(* Logix 5000 project; controller Week1 vendor 1 type 14 code 151 rev 37.11; software revision 37.00 *)

TASK MainTask (continuous, watchdog 500 ms) : MainProgram

MODULES
   Local : vendor 1 type 14 code 151 (Compact 0, rev 37.11)
      Discrete_IO : Embedded (Compact 1, rev 3.1, Output RPI 20 ms)
      Analog_IO : Embedded (Compact 2, rev 1.1, Output RPI 80 ms)
      Counters : Embedded (Compact 3, rev 1.1, Output RPI 20 ms)
END_MODULES

PROGRAM MainProgram   (* main routine MainRoutine *)
VAR
   Cycle_Timer : COUNTER := (PRE := 3, ACC := 3, DN := 1);
   Green_Light : ALIAS FOR Local:1:O.Data.2;
   Green_Pct : REAL := 39.863888;
   Green_Timer : TIMER := (PRE := 300000, ACC := 71755);
   Light_Off : BOOL;
   Logic_Sub : DINT;
   Red_Light : ALIAS FOR Local:1:O.Data.0;
   Red_Pct : REAL := 33.332222;
   Red_Timer : TIMER := (PRE := 300000, ACC := 59998);
   Res_Value : DINT;
   Reset_All : BOOL;
   Reset_PB : ALIAS FOR Local:1:I.Data.0;
   Test_Tag : DINT := 12345;
   Total_Time : DINT;
   Traffic_Timer : TIMER := (PRE := 60000);
   Yellow_Light : ALIAS FOR Local:1:O.Data.1;
   Yellow_Pct : REAL := 8.331667;
   Yellow_Timer : TIMER := (PRE := 300000, ACC := 14997);
END_VAR

ROUTINE MainRoutine   (* ladder *)
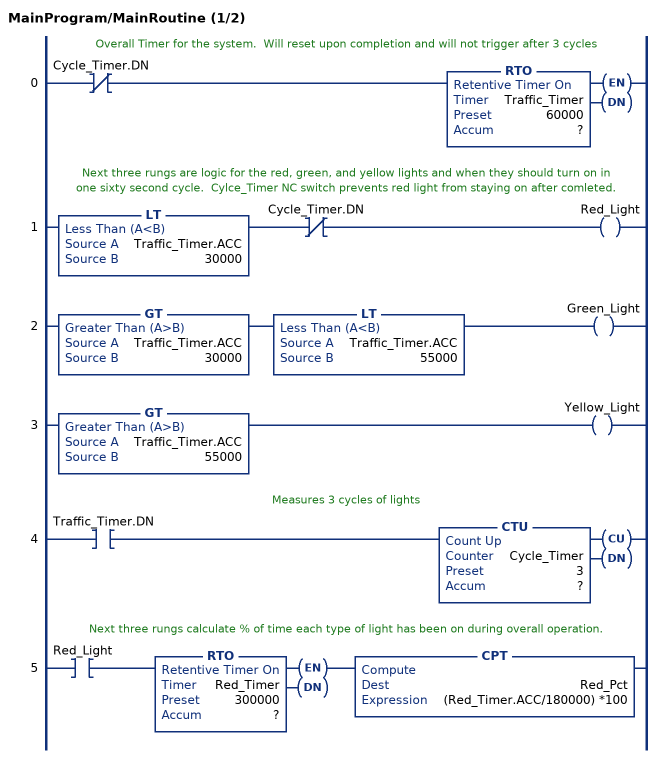
   // Overall Timer for the system.  Will reset upon completion and will not trigger after 3 cycles
   0: XIO(Cycle_Timer.DN)RTO(Traffic_Timer,?,?);
   // Next three rungs are logic for the red, green, and yellow lights and when they should turn on in one sixty second cycle.  Cylce_Timer NC switch prevents red light from staying on after comleted.
   1: LT(Traffic_Timer.ACC,30000)XIO(Cycle_Timer.DN)OTE(Red_Light);
   2: GT(Traffic_Timer.ACC,30000)LT(Traffic_Timer.ACC,55000)OTE(Green_Light);
   3: GT(Traffic_Timer.ACC,55000)OTE(Yellow_Light);
   // Measures 3 cycles of lights
   4: XIC(Traffic_Timer.DN)CTU(Cycle_Timer,?,?);
   // Next three rungs calculate % of time each type of light has been on during overall operation.
   5: XIC(Red_Light)RTO(Red_Timer,?,?)CPT(Red_Pct,(Red_Timer.ACC/180000) *100);
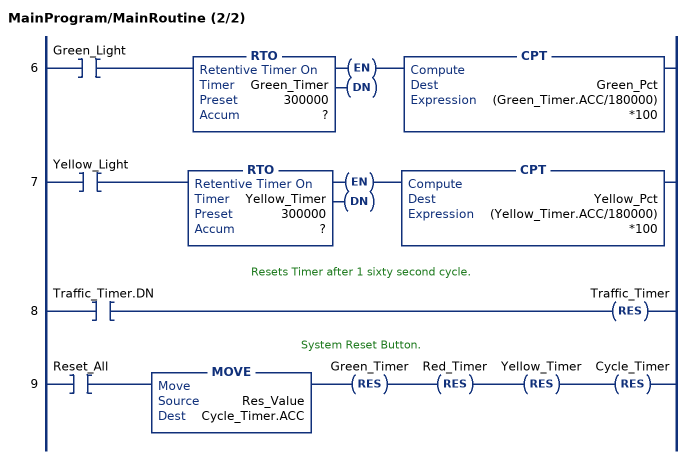
   6: XIC(Green_Light)RTO(Green_Timer,?,?)CPT(Green_Pct,(Green_Timer.ACC/180000) *100);
   7: XIC(Yellow_Light)RTO(Yellow_Timer,?,?)CPT(Yellow_Pct,(Yellow_Timer.ACC/180000) *100);
   // Resets Timer after 1 sixty second cycle.
   8: XIC(Traffic_Timer.DN)RES(Traffic_Timer);
   // System Reset Button.
   9: XIC(Reset_All)MOVE(Res_Value,Cycle_Timer.ACC)RES(Green_Timer)RES(Red_Timer)RES(Yellow_Timer)RES(Cycle_Timer);
END_ROUTINE
END_PROGRAM
